FUNCTION_BLOCK ElectricBoard
VAR_INPUT
END_VAR
VAR_OUTPUT
END_VAR
VAR
	EmergencyBlock: SR;
END_VAR

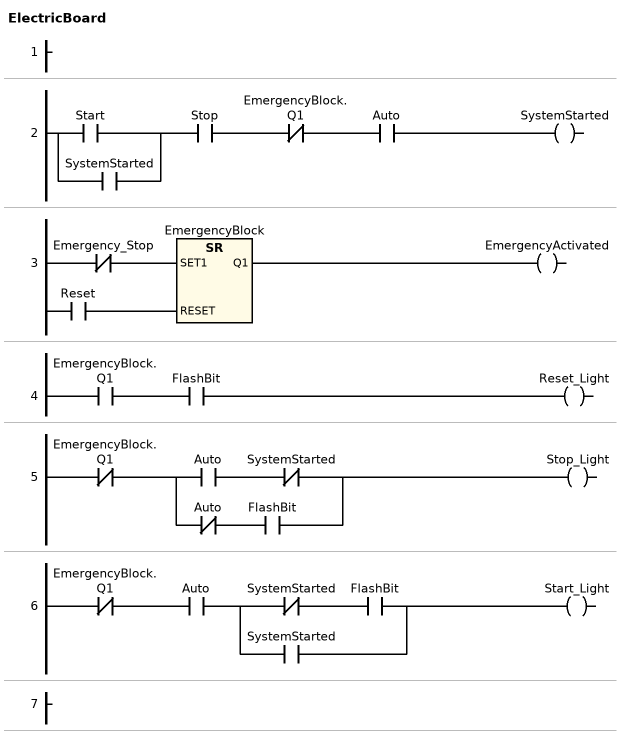
// NETWORK 1

// NETWORK 2
SystemStarted := (Start OR SystemStarted) AND Stop AND NOT EmergencyBlock.Q1 AND Auto;

// NETWORK 3
EmergencyBlock(SET1 := NOT Emergency_Stop, RESET := Reset); // SR
EmergencyActivated := EmergencyBlock.Q1;

// NETWORK 4
Reset_Light := EmergencyBlock.Q1 AND FlashBit;

// NETWORK 5
Stop_Light := NOT EmergencyBlock.Q1 AND (Auto AND NOT SystemStarted OR NOT Auto AND FlashBit);

// NETWORK 6
Start_Light := NOT EmergencyBlock.Q1 AND Auto AND (NOT SystemStarted AND FlashBit OR SystemStarted);

// NETWORK 7

END_FUNCTION_BLOCK

(* stored: Version 1.1.0.1, ProductVersion 3.1.4024.6
   POU ElectricBoard: Id {065d38d7-5a4f-4948-acbb-0327f3e31e43}, SpecialFunc None *)
